(* CoDeSys 2.3.9.59 project: ProgettoSFC_nuovo.pro *)
(* Libraries: STANDARD.LIB, Iecsfc.lib 12.5.98 12:03:00 *)

(* Task configuration *)
TASK Standard (PRIORITY := 0, INTERVAL := T#10ms);
	MAIN
END_TASK

(* Data type *)
TYPE ALTEZZA: (nienteA,basso, alto);
END_TYPE

(* Data type *)
TYPE COLORE: (nienteC,rosso, altro);
END_TYPE

(* Data type *)
TYPE PEZZO :
STRUCT
	Colore : COLORE;
	Altezza : ALTEZZA;
END_STRUCT
END_TYPE

(* Data type *)
TYPE POSTO :
STRUCT
	Presenza :BOOL:=FALSE;
	Pezzo :PEZZO;
END_STRUCT
END_TYPE

(* POU MAIN, SFC *)
PROGRAM MAIN
VAR

(*Variabili Pistone*)
         (*Ingressi*)
	pezzo_magazzino  AT%IX0.0:BOOL;
	pistone_avanti AT%IX0.2:BOOL;
	pistone_indietro AT%IX0.4:BOOL;
         N_pezzi_spinti: INT:=0;
         (*Uscite*)
	pistone_on  AT%QX0.2:BOOL;
        (*TimerPistone*)
	T_pistone: TON;
	mytimepistone: TIME;
	timer_pistone: BOOL;
	reset_timer: BOOL;

(*Variabili Nastro*)
         (*Ingressi*)
	fine_corsa_nastro  AT%IX0.6:BOOL;
         (*Uscite*)
	nastro_on  AT%QX0.0:BOOL;


(*Variabili Giostra*)
        Giostra: ARRAY[0..7] OF POSTO;
	i: INT :=0;

        (*Ingressi*)
        giostra_busy AT %IX6.1: BOOL;

        sensore_colore AT %IX2.1: BOOL;

        trapano_basso AT %IX2.5: BOOL ;
        trapano_alto AT %IX2.3: BOOL;

        tastatore_basso AT %IX5.3: BOOL;
        tastatore_alto AT %IX2.7: BOOL;

        pennarello_alto AT %IX5.4: BOOL;
        pennarello_basso AT %IX5.5: BOOL;

        pistone_PT5_avanti AT %IX5.0: BOOL;
        pistone_PT5_indietro AT %IX5.1: BOOL;

        pistone_PT6_avanti AT %IX5.7: BOOL;
        pistone_PT6_indietro AT %IX5.6: BOOL;

        pezzo_baia AT %IX5.2: BOOL;

        (*Uscite*)
        movimento_giostra AT %QX3.4: BOOL;

        trapano_on AT %QX3.7:BOOL;
        trapano_down AT %QX7.0: BOOL;

        tastatore_down AT %QX3.6: BOOL;

        pennarello_down AT %QX3.3: BOOL;

        pistone_PT5_on AT %QX3.1:BOOL ;
        pistone_PT6_on AT%QX3.5: BOOL;

	T_giostra: TON;
         mytimegiostra: TIME;
	timer_giostra: BOOL;
	reset_timer_giostra: BOOL;

	T_trapano: TON;
	mytimetrapano: TIME;
	timer_trapano: BOOL;
	reset_timer_trapano: BOOL;

	(*T_p1: TON;
	mytimep1: TIME;
	timer_p1: BOOL;
	reset_timer_p1: BOOL;*)

	T_pennarello: TON;
	mytimepennarello: TIME;
	timer_pennarello: BOOL;
	reset_timer_pennarello: BOOL;

	mytimep1: TIME;
	T_p1: TON;
	reset_timer_p1: BOOL;
	timer_p1: BOOL;
	reset_timer_tastatore: BOOL;
	mytimetastatore: TIME;
	T_tastatore: TON;
	timer_tastatore: BOOL;
	j: INT;
	condizione: BOOL;
END_VAR
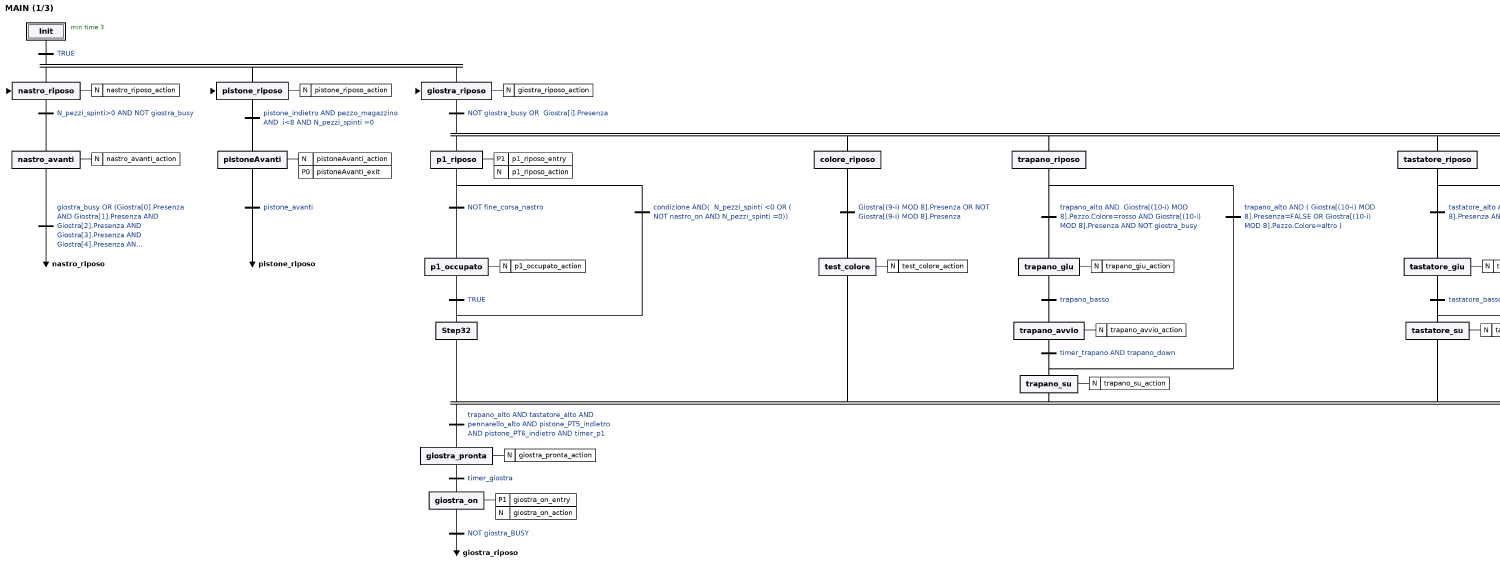
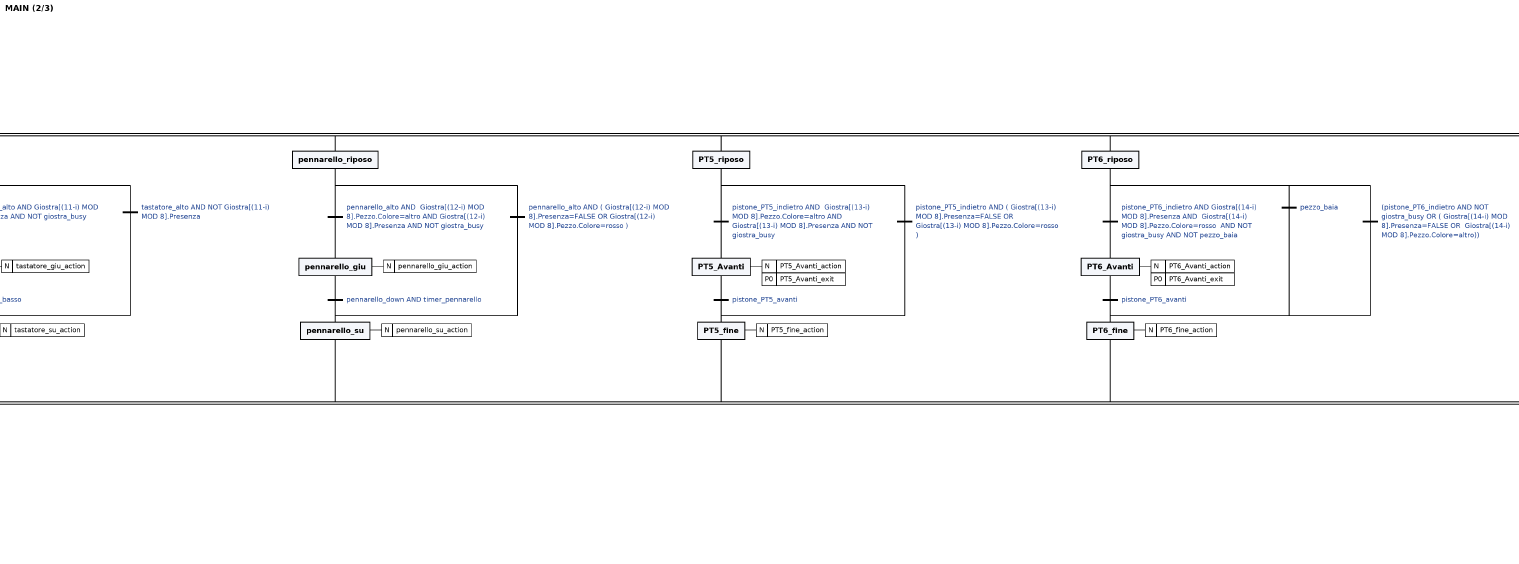
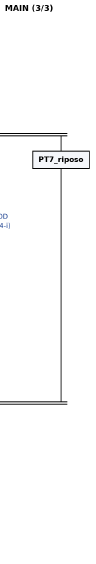
INITIAL_STEP Init: (* min time 3 *)
END_STEP
TRANSITION FROM Init TO (nastro_riposo, pistone_riposo, giostra_riposo) := TRUE;
END_TRANSITION
STEP nastro_riposo:
	nastro_riposo_action(N);
END_STEP
TRANSITION FROM nastro_riposo TO nastro_avanti := N_pezzi_spinti>0 AND NOT giostra_busy;
END_TRANSITION
STEP pistone_riposo:
	pistone_riposo_action(N);
END_STEP
TRANSITION FROM pistone_riposo TO pistoneAvanti := pistone_indietro AND pezzo_magazzino  AND  i<8 AND N_pezzi_spinti =0;
END_TRANSITION
STEP giostra_riposo:
	giostra_riposo_action(N);
END_STEP
TRANSITION FROM giostra_riposo TO (p1_riposo, colore_riposo, trapano_riposo, tastatore_riposo, pennarello_riposo, PT5_riposo, PT6_riposo, PT7_riposo) := NOT giostra_busy OR  Giostra[i].Presenza;
END_TRANSITION
STEP p1_riposo:
	p1_riposo_entry(P1);
	p1_riposo_action(N);
END_STEP
TRANSITION FROM p1_riposo TO p1_occupato := NOT fine_corsa_nastro;
END_TRANSITION
TRANSITION FROM p1_riposo TO Step32 := condizione AND(  N_pezzi_spinti <0 OR ( NOT nastro_on AND N_pezzi_spinti =0));
END_TRANSITION
STEP p1_occupato:
	p1_occupato_action(N);
END_STEP
TRANSITION FROM p1_occupato TO Step32 := TRUE;
END_TRANSITION
STEP Step32:
END_STEP
STEP colore_riposo:
END_STEP
TRANSITION FROM colore_riposo TO test_colore := Giostra[(9-i) MOD 8].Presenza OR NOT Giostra[(9-i) MOD 8].Presenza;
END_TRANSITION
STEP test_colore:
	test_colore_action(N);
END_STEP
STEP trapano_riposo:
END_STEP
TRANSITION FROM trapano_riposo TO trapano_giu := trapano_alto AND  Giostra[(10-i) MOD 8].Pezzo.Colore=rosso AND Giostra[(10-i) MOD 8].Presenza AND NOT giostra_busy;
END_TRANSITION
TRANSITION FROM trapano_riposo TO trapano_su := trapano_alto AND ( Giostra[(10-i) MOD 8].Presenza=FALSE OR Giostra[(10-i) MOD 8].Pezzo.Colore=altro );
END_TRANSITION
STEP trapano_giu:
	trapano_giu_action(N);
END_STEP
TRANSITION FROM trapano_giu TO trapano_avvio := trapano_basso;
END_TRANSITION
STEP trapano_avvio:
	trapano_avvio_action(N);
END_STEP
TRANSITION FROM trapano_avvio TO trapano_su := timer_trapano AND trapano_down;
END_TRANSITION
STEP trapano_su:
	trapano_su_action(N);
END_STEP
STEP tastatore_riposo:
END_STEP
TRANSITION FROM tastatore_riposo TO tastatore_giu := tastatore_alto AND Giostra[(11-i) MOD 8].Presenza AND NOT giostra_busy;
END_TRANSITION
TRANSITION FROM tastatore_riposo TO tastatore_su := tastatore_alto AND NOT Giostra[(11-i) MOD 8].Presenza;
END_TRANSITION
STEP tastatore_giu:
	tastatore_giu_action(N);
END_STEP
TRANSITION FROM tastatore_giu TO tastatore_su := tastatore_basso;
END_TRANSITION
STEP tastatore_su:
	tastatore_su_action(N);
END_STEP
STEP pennarello_riposo:
END_STEP
TRANSITION FROM pennarello_riposo TO pennarello_giu := pennarello_alto AND  Giostra[(12-i) MOD 8].Pezzo.Colore=altro AND Giostra[(12-i) MOD 8].Presenza AND NOT giostra_busy;
END_TRANSITION
TRANSITION FROM pennarello_riposo TO pennarello_su := pennarello_alto AND ( Giostra[(12-i) MOD 8].Presenza=FALSE OR Giostra[(12-i) MOD 8].Pezzo.Colore=rosso );
END_TRANSITION
STEP pennarello_giu:
	pennarello_giu_action(N);
END_STEP
TRANSITION FROM pennarello_giu TO pennarello_su := pennarello_down AND timer_pennarello;
END_TRANSITION
STEP pennarello_su:
	pennarello_su_action(N);
END_STEP
STEP PT5_riposo:
END_STEP
TRANSITION FROM PT5_riposo TO PT5_Avanti := pistone_PT5_indietro AND  Giostra[(13-i) MOD 8].Pezzo.Colore=altro AND Giostra[(13-i) MOD 8].Presenza AND NOT giostra_busy;
END_TRANSITION
TRANSITION FROM PT5_riposo TO PT5_fine := pistone_PT5_indietro AND ( Giostra[(13-i) MOD 8].Presenza=FALSE OR Giostra[(13-i) MOD 8].Pezzo.Colore=rosso );
END_TRANSITION
STEP PT5_Avanti:
	PT5_Avanti_action(N);
	PT5_Avanti_exit(P0);
END_STEP
TRANSITION FROM PT5_Avanti TO PT5_fine := pistone_PT5_avanti;
END_TRANSITION
STEP PT5_fine:
	PT5_fine_action(N);
END_STEP
STEP PT6_riposo:
END_STEP
TRANSITION FROM PT6_riposo TO PT6_Avanti := pistone_PT6_indietro AND Giostra[(14-i) MOD 8].Presenza AND  Giostra[(14-i) MOD 8].Pezzo.Colore=rosso  AND NOT giostra_busy AND NOT pezzo_baia;
END_TRANSITION
TRANSITION FROM PT6_riposo TO PT6_fine := pezzo_baia;
END_TRANSITION
TRANSITION FROM PT6_riposo TO PT6_fine := (pistone_PT6_indietro AND NOT giostra_busy OR ( Giostra[(14-i) MOD 8].Presenza=FALSE OR  Giostra[(14-i) MOD 8].Pezzo.Colore=altro));
END_TRANSITION
STEP PT6_Avanti:
	PT6_Avanti_action(N);
	PT6_Avanti_exit(P0);
END_STEP
TRANSITION FROM PT6_Avanti TO PT6_fine := pistone_PT6_avanti;
END_TRANSITION
STEP PT6_fine:
	PT6_fine_action(N);
END_STEP
STEP PT7_riposo:
END_STEP
TRANSITION FROM (Step32, test_colore, trapano_su, tastatore_su, pennarello_su, PT5_fine, PT6_fine, PT7_riposo) TO giostra_pronta := trapano_alto AND tastatore_alto AND pennarello_alto AND pistone_PT5_indietro AND pistone_PT6_indietro AND timer_p1;
END_TRANSITION
STEP giostra_pronta:
	giostra_pronta_action(N);
END_STEP
TRANSITION FROM giostra_pronta TO giostra_on := timer_giostra;
END_TRANSITION
STEP giostra_on:
	giostra_on_entry(P1);
	giostra_on_action(N);
END_STEP
TRANSITION FROM giostra_on TO giostra_riposo := NOT giostra_BUSY;
END_TRANSITION
STEP pistoneAvanti:
	pistoneAvanti_action(N);
	pistoneAvanti_exit(P0);
END_STEP
TRANSITION FROM pistoneAvanti TO pistone_riposo := pistone_avanti;
END_TRANSITION
STEP nastro_avanti:
	nastro_avanti_action(N);
END_STEP
TRANSITION FROM nastro_avanti TO nastro_riposo := giostra_busy OR (Giostra[0].Presenza AND Giostra[1].Presenza AND Giostra[2].Presenza AND Giostra[3].Presenza AND Giostra[4].Presenza AND Giostra[5].Presenza AND Giostra[6].Presenza AND Giostra[7].Presenza);
END_TRANSITION

ACTION nastro_riposo_action:
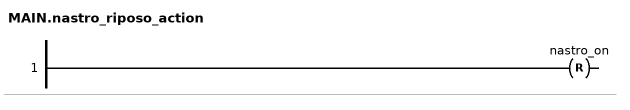
_LD_ (* Ladder Diagram *)
NETWORK 1
	* --- (R nastro_on)
_END_LD_
(* the same logic as Structured Text *)
(* Network 1 *)
nastro_on := FALSE;
END_ACTION

ACTION pistone_riposo_action:
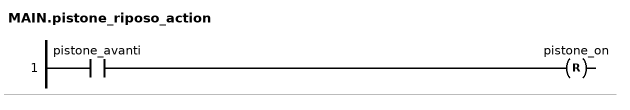
_LD_ (* Ladder Diagram *)
NETWORK 1
	[pistone_avanti] --- (R pistone_on)
_END_LD_
(* the same logic as Structured Text *)
(* Network 1 *)
IF pistone_avanti THEN pistone_on := FALSE; END_IF;
END_ACTION

ACTION giostra_riposo_action:
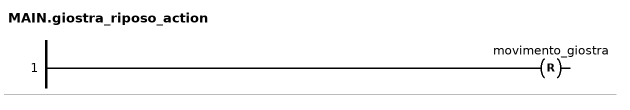
_LD_ (* Ladder Diagram *)
NETWORK 1
	* --- (R movimento_giostra)
_END_LD_
(* the same logic as Structured Text *)
(* Network 1 *)
movimento_giostra := FALSE;
END_ACTION

ACTION p1_riposo_entry:
FOR j:=0 TO 7 BY 1  DO
IF(Giostra[j].Presenza) THEN condizione:=TRUE;
EXIT;
ELSE condizione:=FALSE;
END_IF;
END_FOR;
END_ACTION

ACTION p1_riposo_action:
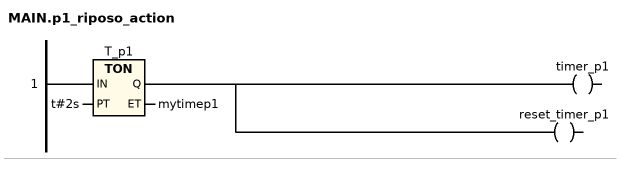
_LD_ (* Ladder Diagram *)
NETWORK 1
	T_p1:TON(IN: *, PT: t#2s, ET => mytimep1) --- (timer_p1) (reset_timer_p1)
_END_LD_
(* the same logic as Structured Text *)
(* Network 1 *)
T_p1(IN := TRUE, PT := t#2s);
mytimep1 := T_p1.ET;
timer_p1 := T_p1.Q;
reset_timer_p1 := T_p1.Q;
END_ACTION

ACTION p1_occupato_action:
Giostra[(8-i)MOD 8].Presenza:=TRUE;
N_pezzi_spinti:=N_pezzi_spinti-1;
END_ACTION

ACTION test_colore_action:
IF (sensore_colore=TRUE) THEN
Giostra[(9-i) MOD 8].Pezzo.Colore:=rosso;
ELSE
Giostra[(9-i) MOD 8].Pezzo.Colore:=altro;
END_IF
END_ACTION

ACTION trapano_giu_action:
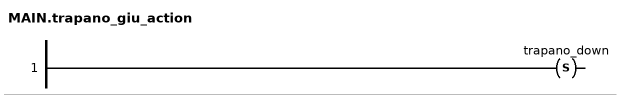
_LD_ (* Ladder Diagram *)
NETWORK 1
	* --- (S trapano_down)
_END_LD_
(* the same logic as Structured Text *)
(* Network 1 *)
trapano_down := TRUE;
END_ACTION

ACTION trapano_avvio_action:
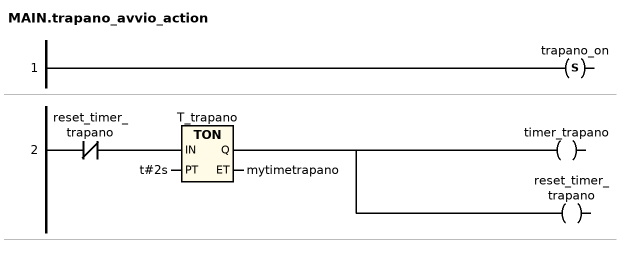
_LD_ (* Ladder Diagram *)
NETWORK 1
	* --- (S trapano_on)
NETWORK 2
	[/reset_timer_trapano] - T_trapano:TON(IN: *, PT: t#2s, ET => mytimetrapano) --- (timer_trapano) (reset_timer_trapano)
_END_LD_
(* the same logic as Structured Text *)
(* Network 1 *)
trapano_on := TRUE;
(* Network 2 *)
T_trapano(IN := NOT reset_timer_trapano, PT := t#2s);
mytimetrapano := T_trapano.ET;
timer_trapano := T_trapano.Q;
reset_timer_trapano := T_trapano.Q;
END_ACTION

ACTION trapano_su_action:
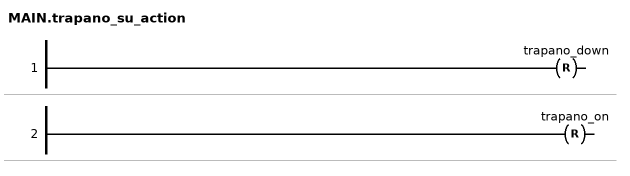
_LD_ (* Ladder Diagram *)
NETWORK 1
	* --- (R trapano_down)
NETWORK 2
	* --- (R trapano_on)
_END_LD_
(* the same logic as Structured Text *)
(* Network 1 *)
trapano_down := FALSE;
(* Network 2 *)
trapano_on := FALSE;
END_ACTION

ACTION tastatore_giu_action:
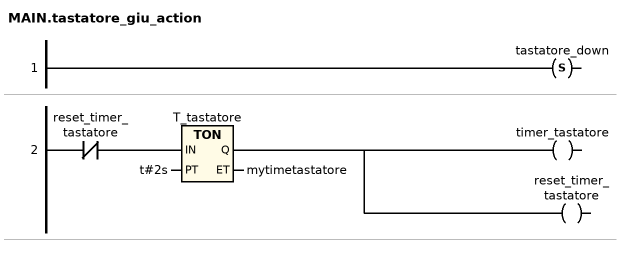
_LD_ (* Ladder Diagram *)
NETWORK 1
	* --- (S tastatore_down)
NETWORK 2
	[/reset_timer_tastatore] - T_tastatore:TON(IN: *, PT: t#2s, ET => mytimetastatore) --- (timer_tastatore) (reset_timer_tastatore)
_END_LD_
(* the same logic as Structured Text *)
(* Network 1 *)
tastatore_down := TRUE;
(* Network 2 *)
T_tastatore(IN := NOT reset_timer_tastatore, PT := t#2s);
mytimetastatore := T_tastatore.ET;
timer_tastatore := T_tastatore.Q;
reset_timer_tastatore := T_tastatore.Q;
END_ACTION

ACTION tastatore_su_action:
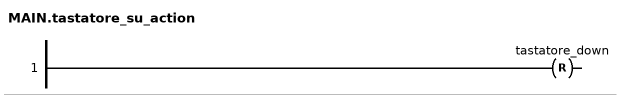
_LD_ (* Ladder Diagram *)
NETWORK 1
	* --- (R tastatore_down)
_END_LD_
(* the same logic as Structured Text *)
(* Network 1 *)
tastatore_down := FALSE;
END_ACTION

ACTION pennarello_giu_action:
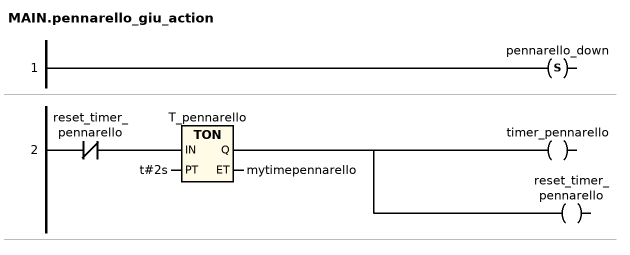
_LD_ (* Ladder Diagram *)
NETWORK 1
	* --- (S pennarello_down)
NETWORK 2
	[/reset_timer_pennarello] - T_pennarello:TON(IN: *, PT: t#2s, ET => mytimepennarello) --- (timer_pennarello) (reset_timer_pennarello)
_END_LD_
(* the same logic as Structured Text *)
(* Network 1 *)
pennarello_down := TRUE;
(* Network 2 *)
T_pennarello(IN := NOT reset_timer_pennarello, PT := t#2s);
mytimepennarello := T_pennarello.ET;
timer_pennarello := T_pennarello.Q;
reset_timer_pennarello := T_pennarello.Q;
END_ACTION

ACTION pennarello_su_action:
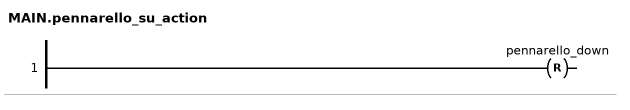
_LD_ (* Ladder Diagram *)
NETWORK 1
	* --- (R pennarello_down)
_END_LD_
(* the same logic as Structured Text *)
(* Network 1 *)
pennarello_down := FALSE;
END_ACTION

ACTION PT5_Avanti_action:
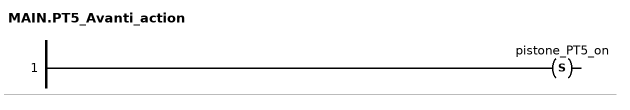
_LD_ (* Ladder Diagram *)
NETWORK 1
	* --- (S pistone_PT5_on)
_END_LD_
(* the same logic as Structured Text *)
(* Network 1 *)
pistone_PT5_on := TRUE;
END_ACTION

ACTION PT5_Avanti_exit:
Giostra[(13-i) MOD 8].Presenza:=FALSE;
Giostra[(13-i) MOD 8].Pezzo.Colore:=nienteC;
END_ACTION

ACTION PT5_fine_action:
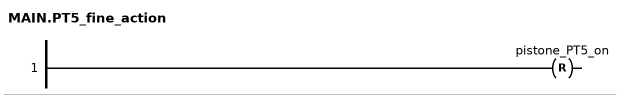
_LD_ (* Ladder Diagram *)
NETWORK 1
	* --- (R pistone_PT5_on)
_END_LD_
(* the same logic as Structured Text *)
(* Network 1 *)
pistone_PT5_on := FALSE;
END_ACTION

ACTION PT6_Avanti_action:
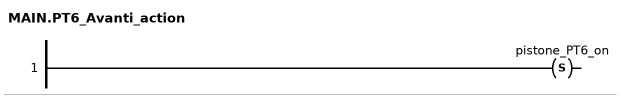
_LD_ (* Ladder Diagram *)
NETWORK 1
	* --- (S pistone_PT6_on)
_END_LD_
(* the same logic as Structured Text *)
(* Network 1 *)
pistone_PT6_on := TRUE;
END_ACTION

ACTION PT6_Avanti_exit:
Giostra[(14-i) MOD 8].Presenza:=FALSE;
Giostra[(14-i) MOD 8].Pezzo.Colore:=nienteC;
END_ACTION

ACTION PT6_fine_action:
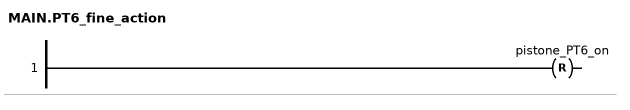
_LD_ (* Ladder Diagram *)
NETWORK 1
	* --- (R pistone_PT6_on)
_END_LD_
(* the same logic as Structured Text *)
(* Network 1 *)
pistone_PT6_on := FALSE;
END_ACTION

ACTION giostra_pronta_action:
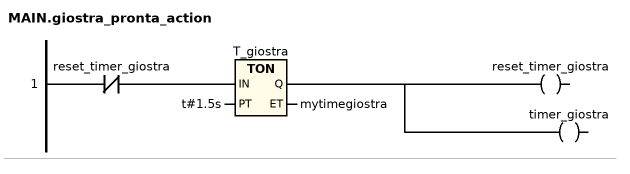
_LD_ (* Ladder Diagram *)
NETWORK 1
	[/reset_timer_giostra] - T_giostra:TON(IN: *, PT: t#1.5s, ET => mytimegiostra) --- (reset_timer_giostra) (timer_giostra)
_END_LD_
(* the same logic as Structured Text *)
(* Network 1 *)
T_giostra(IN := NOT reset_timer_giostra, PT := t#1.5s);
mytimegiostra := T_giostra.ET;
reset_timer_giostra := T_giostra.Q;
timer_giostra := T_giostra.Q;
END_ACTION

ACTION giostra_on_entry:
IF( i=7) THEN i:=0;
ELSE i:=i+1;
END_IF
END_ACTION

ACTION giostra_on_action:
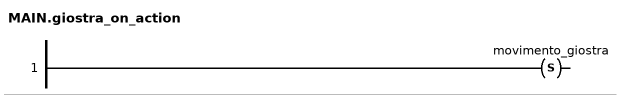
_LD_ (* Ladder Diagram *)
NETWORK 1
	* --- (S movimento_giostra)
_END_LD_
(* the same logic as Structured Text *)
(* Network 1 *)
movimento_giostra := TRUE;
END_ACTION

ACTION pistoneAvanti_action:
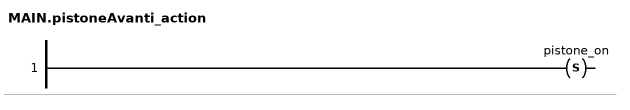
_LD_ (* Ladder Diagram *)
NETWORK 1
	* --- (S pistone_on)
_END_LD_
(* the same logic as Structured Text *)
(* Network 1 *)
pistone_on := TRUE;
END_ACTION

ACTION pistoneAvanti_exit:
N_pezzi_spinti:=N_pezzi_spinti+1;
END_ACTION

ACTION nastro_avanti_action:
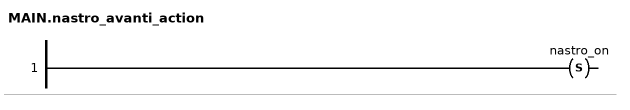
_LD_ (* Ladder Diagram *)
NETWORK 1
	* --- (S nastro_on)
_END_LD_
(* the same logic as Structured Text *)
(* Network 1 *)
nastro_on := TRUE;
END_ACTION
END_PROGRAM
